Fanuc KAREL source: kb00026.KL

-- PROVISIONAL review KL for V1013-1; original PC SHA256 2e1fa0f733bc6034aeb54c5fd695a86a8ceaf42add2e93eaced9cf03cf5f60f4
-- Incomplete behavior may be omitted. Consult companion uncertainty JSON. Do not deploy.
PROGRAM KB00026
%NOLOCKGROUP
BEGIN
  -- UNRESOLVED_PC offsets 5-12; opcodes 9D,23
  -- UNRESOLVED_PC offsets 17-24; opcodes 9D,23
  -- UNRESOLVED_PC offsets 29-36; opcodes 9D,23
  -- UNRESOLVED_PC offsets 41-63; opcodes 27,22,22,22,31
  -- UNRESOLVED_PC offsets 68-72; opcodes 7F
END KB00026
